Fanuc KAREL source: kt00212.KL

PROGRAM KT00212
%STACKSIZE=65535
%PRIORITY=65535
%NOLOCKGROUP
VAR
Y1 : ARRAY[2] OF BYTE
I2 : INTEGER
OUT : INTEGER
BEGIN
Y1[1]=2
I2=3
-- UNRESOLVED_PC line 10 opcodes [22 9D 33 B1 21 46 23] marker_code=35
END KT00212
